FUNCTION_BLOCK "ST10_Flow3_A1RotaryShaftScan"
VAR_INPUT
  iSysInface : "RCS_SysComInterface_V1";
END_VAR
VAR_IN_OUT
  ioPM_Inface : "RCS_PMInterface_V1";
  ioStatus : Int;
END_VAR
VAR
  sCtrlMode : "SysFlowCtrlGraph";
  sUpdMES_Data : Bool;
  "工件放行中" : Bool;
  "前站站号" : UInt;
  "本站站号" : UInt;
  "弹窗Temp" : Array[1..10] of Int;
  AlarmID : Int;
  TON : Array[0..10] of TON_TIME;
  TOF : Array[0..10] of TOF_TIME;
  sUP : Array[0..10] of Bool;
  "更新RFID完成" : Bool;
  RT_DATA : G7_RTDataPlus_V6;
  Trans1 : G7_TransitionPlus_V6;
  Trans2 : G7_TransitionPlus_V6;
  Trans3 : G7_TransitionPlus_V6;
  Trans325 : G7_TransitionPlus_V6;
  Trans10 : G7_TransitionPlus_V6;
  Trans7 : G7_TransitionPlus_V6;
  Trans102 : G7_TransitionPlus_V6;
  Trans8 : G7_TransitionPlus_V6;
  Trans12 : G7_TransitionPlus_V6;
  Offline : G7_TransitionPlus_V6;
  Trans200 : G7_TransitionPlus_V6;
  Empty : G7_TransitionPlus_V6;
  Trans266 : G7_TransitionPlus_V6;
  Trans11 : G7_TransitionPlus_V6;
  Trans249 : G7_TransitionPlus_V6;
  Trans283 : G7_TransitionPlus_V6;
  Trans199 : G7_TransitionPlus_V6;
  HavePart : G7_TransitionPlus_V6;
  Trans303 : G7_TransitionPlus_V6;
  Trans304 : G7_TransitionPlus_V6;
  Trans145 : G7_TransitionPlus_V6;
  Trans146 : G7_TransitionPlus_V6;
  Trans147 : G7_TransitionPlus_V6;
  Trans201 : G7_TransitionPlus_V6;
  Trans202 : G7_TransitionPlus_V6;
  ReadNG : G7_TransitionPlus_V6;
  ReadOK : G7_TransitionPlus_V6;
  Trans205 : G7_TransitionPlus_V6;
  Trans203 : G7_TransitionPlus_V6;
  Trans204 : G7_TransitionPlus_V6;
  ReadNG_2 : G7_TransitionPlus_V6;
  Trans206 : G7_TransitionPlus_V6;
  ReadOK_2 : G7_TransitionPlus_V6;
  Trans211 : G7_TransitionPlus_V6;
  Trans212 : G7_TransitionPlus_V6;
  Trans213 : G7_TransitionPlus_V6;
  Trans207 : G7_TransitionPlus_V6;
  Trans208 : G7_TransitionPlus_V6;
  ReadNG_3 : G7_TransitionPlus_V6;
  ReadOK_3 : G7_TransitionPlus_V6;
  Trans209 : G7_TransitionPlus_V6;
  Trans210 : G7_TransitionPlus_V6;
  Trans214 : G7_TransitionPlus_V6;
  ReadNG_4 : G7_TransitionPlus_V6;
  ReadOK_4 : G7_TransitionPlus_V6;
  Trans215 : G7_TransitionPlus_V6;
  Trans216 : G7_TransitionPlus_V6;
  Trans217 : G7_TransitionPlus_V6;
  ReadNG_5 : G7_TransitionPlus_V6;
  ReadOK_5 : G7_TransitionPlus_V6;
  Trans218 : G7_TransitionPlus_V6;
  Trans219 : G7_TransitionPlus_V6;
  Trans220 : G7_TransitionPlus_V6;
  ReadNG_6 : G7_TransitionPlus_V6;
  ReadOK_6 : G7_TransitionPlus_V6;
  Trans221 : G7_TransitionPlus_V6;
  Trans222 : G7_TransitionPlus_V6;
  Trans223 : G7_TransitionPlus_V6;
  ReadNG_7 : G7_TransitionPlus_V6;
  ReadOK_7 : G7_TransitionPlus_V6;
  Trans225 : G7_TransitionPlus_V6;
  Trans226 : G7_TransitionPlus_V6;
  Trans227 : G7_TransitionPlus_V6;
  ReadNG_8 : G7_TransitionPlus_V6;
  ReadOK_8 : G7_TransitionPlus_V6;
  Trans246 : G7_TransitionPlus_V6;
  Trans230 : G7_TransitionPlus_V6;
  Trans247 : G7_TransitionPlus_V6;
  Trans248 : G7_TransitionPlus_V6;
  Trans250 : G7_TransitionPlus_V6;
  Trans251 : G7_TransitionPlus_V6;
  Trans252 : G7_TransitionPlus_V6;
  Trans253 : G7_TransitionPlus_V6;
  Trans254 : G7_TransitionPlus_V6;
  Trans257 : G7_TransitionPlus_V6;
  Trans261 : G7_TransitionPlus_V6;
  Online : G7_TransitionPlus_V6;
  Trans259 : G7_TransitionPlus_V6;
  Trans260 : G7_TransitionPlus_V6;
  Trans14 : G7_TransitionPlus_V6;
  Trans15 : G7_TransitionPlus_V6;
  Trans264 : G7_TransitionPlus_V6;
  Trans265 : G7_TransitionPlus_V6;
  Trans307 : G7_TransitionPlus_V6;
  Trans308 : G7_TransitionPlus_V6;
  Trans315 : G7_TransitionPlus_V6;
  Trans310 : G7_TransitionPlus_V6;
  Trans311 : G7_TransitionPlus_V6;
  Trans312 : G7_TransitionPlus_V6;
  Trans313 : G7_TransitionPlus_V6;
  Trans610 : G7_TransitionPlus_V6;
  Trans314 : G7_TransitionPlus_V6;
  Trans16 : G7_TransitionPlus_V6;
  Trans317 : G7_TransitionPlus_V6;
  Trans318 : G7_TransitionPlus_V6;
  Trans319 : G7_TransitionPlus_V6;
  Trans320 : G7_TransitionPlus_V6;
  Trans316 : G7_TransitionPlus_V6;
  Trans322 : G7_TransitionPlus_V6;
  Trans412 : G7_TransitionPlus_V6;
  Trans600 : G7_TransitionPlus_V6;
  Trans699 : G7_TransitionPlus_V6;
  Trans613 : G7_TransitionPlus_V6;
  Alarm : G7_TransitionPlus_V6;
  F3_Initial : G7_StepPlus_V6;
  S2 : G7_StepPlus_V6;
  S3 : G7_StepPlus_V6;
  "ServoReady?" : G7_StepPlus_V6;
  S5_MESInitial : G7_StepPlus_V6;
  WaitRobotInitialFinish : G7_StepPlus_V6;
  "Servo returns to initial Pos" : G7_StepPlus_V6;
  S10_InitialFinish : G7_StepPlus_V6;
  "Servo returns to initial Pos_1" : G7_StepPlus_V6;
  "MES OK" : G7_StepPlus_V6;
  ProcessStart : G7_StepPlus_V6;
  "Determine product status" : G7_StepPlus_V6;
  CheckMachineStatus : G7_StepPlus_V6;
  "Normal mode" : G7_StepPlus_V6;
  "ProcessStart,CTStart" : G7_StepPlus_V6;
  "Request robot put" : G7_StepPlus_V6;
  RobotPutPartFinish : G7_StepPlus_V6;
  PartStatusOK : G7_StepPlus_V6;
  StatusAlarm : G7_StepPlus_V6;
  PartStatusError : G7_StepPlus_V6;
  NoPart : G7_StepPlus_V6;
  "Wait  robot finish task" : G7_StepPlus_V6;
  "Wait robot finish task" : G7_StepPlus_V6;
  "Wait robot in safety area" : G7_StepPlus_V6;
  "Rotary code reading" : G7_StepPlus_V6;
  "Start 1st reading" : G7_StepPlus_V6;
  "Check reader Ready" : G7_StepPlus_V6;
  "Wait reading complete" : G7_StepPlus_V6;
  "Servo returns to Scan2 Pos" : G7_StepPlus_V6;
  "Start 2st reading" : G7_StepPlus_V6;
  "Check reader Ready_1" : G7_StepPlus_V6;
  "Wait reading complete_1" : G7_StepPlus_V6;
  Step208 : G7_StepPlus_V6;
  "Read OK" : G7_StepPlus_V6;
  "Servo returns to Scan3 Pos" : G7_StepPlus_V6;
  "Start 3st reading" : G7_StepPlus_V6;
  "Check reader Ready_2" : G7_StepPlus_V6;
  "Wait reading complete_3" : G7_StepPlus_V6;
  "Servo returns to Scan4 Pos" : G7_StepPlus_V6;
  "Start 4st reading_1" : G7_StepPlus_V6;
  "Check reader Ready_3" : G7_StepPlus_V6;
  "Wait reading complete_4" : G7_StepPlus_V6;
  "Servo returns to Scan5 Pos" : G7_StepPlus_V6;
  "Start 5st reading" : G7_StepPlus_V6;
  "Check reader Ready_4" : G7_StepPlus_V6;
  "Wait reading complete_5" : G7_StepPlus_V6;
  "Servo returns to Scan6Pos" : G7_StepPlus_V6;
  "Start 6st reading" : G7_StepPlus_V6;
  "Check reader Ready_5" : G7_StepPlus_V6;
  "Wait reading complete_6" : G7_StepPlus_V6;
  "Servo returns to Scan7Pos" : G7_StepPlus_V6;
  "Start 7st reading" : G7_StepPlus_V6;
  "Check reader Ready_6" : G7_StepPlus_V6;
  "Wait reading complete_7" : G7_StepPlus_V6;
  "Servo returns to Scan8Pos" : G7_StepPlus_V6;
  "Start 8st reading" : G7_StepPlus_V6;
  "Check reader Ready_7" : G7_StepPlus_V6;
  "Wait reading complete_8" : G7_StepPlus_V6;
  "Read NG" : G7_StepPlus_V6;
  NG_Status : G7_StepPlus_V6;
  OKStatus : G7_StepPlus_V6;
  CheckPartExist : G7_StepPlus_V6;
  PartStatus : G7_StepPlus_V6;
  MES : G7_StepPlus_V6;
  ResetMesCheckRequest : G7_StepPlus_V6;
  ResetMesUnloadRequest_1 : G7_StepPlus_V6;
  "Prepare MES CheckData" : G7_StepPlus_V6;
  "Prepare MES CheckData_1" : G7_StepPlus_V6;
  MESCheckRequest : G7_StepPlus_V6;
  MESSaveRequest_1 : G7_StepPlus_V6;
  "MES NG" : G7_StepPlus_V6;
  MESOverTime : G7_StepPlus_V6;
  ok : G7_StepPlus_V6;
  Bypass : G7_StepPlus_V6;
  MESOverTime_1 : G7_StepPlus_V6;
  ResultNG : G7_StepPlus_V6;
  MESResultFinish : G7_StepPlus_V6;
  Step314 : G7_StepPlus_V6;
  ok_1 : G7_StepPlus_V6;
  "Check OK" : G7_StepPlus_V6;
  "Check NG" : G7_StepPlus_V6;
  "Request robot pick" : G7_StepPlus_V6;
  RobotPick : G7_StepPlus_V6;
  ProcessFinsh : G7_StepPlus_V6;
END_VAR
VAR_TEMP
  Tempresult : USInt;
  "本站站号乘10" : UInt;
END_VAR
BEGIN
  // Původní jazyk: GRAPH
  // Zdroj XML: EXPORT/Program blocks/OP010/03_Auto/A1_TableLoad&Scan/ST10_Flow3_A1RotaryShaftScan.xml
  // (Nebylo nalezeno StructuredText/FlgNet/StatementList; logika může být v GRAPH nebo v nepodporované reprezentaci.)
END_FUNCTION_BLOCK
